FUNCTION FC_Add : DINT
VAR_INPUT
    nA : DINT;
    nB : DINT;
END_VAR
VAR
    nResult : DINT;
END_VAR

nResult := nA + nB;
FC_Add := nResult;

END_FUNCTION

(* stored: Version 1.1.0.1
   POU FC_Add: Id {22222222-2222-2222-2222-222222222222}, SpecialFunc None *)
